PROGRAM P_Demo_FB_HVACHeatingCurve
VAR
    fb : FB_HVACHeatingCurve;                            // 被演示 FB 实例
    eDataSecurityType_in : E_HVACDataSecurityType ;
    bSetDefault_in : BOOL := FALSE;
    rOutsideTempDamped_in : REAL := 0.0;
    bDayOperation_in : BOOL := FALSE;
    bReset_in : BOOL := FALSE;
    rMinTemp_io : REAL := 0.0;
    rMaxTemp_io : REAL := 0.0;
    rNightSetback_io : REAL := 0.0;
    rTempSetpoint_Y1_io : REAL := 0.0;
    rTempSetpoint_Y2_io : REAL := 0.0;
    rTempSetpoint_Y3_io : REAL := 0.0;
    rTempSetpoint_Y4_io : REAL := 0.0;
    rOutsideTemp_X1_io : REAL := 0.0;
    rOutsideTemp_X2_io : REAL := 0.0;
    rOutsideTemp_X3_io : REAL := 0.0;
    rOutsideTemp_X4_io : REAL := 0.0;
    rTempSetpoint_out : REAL;
    bInvalidParameter_out : BOOL;
END_VAR

// ============================================================================
// Tc2_HVAC.FB_HVACHeatingCurve 演示程序
// ============================================================================
// 场景：把本 FB 实例化到一个 PLC 程序里，每周期单次调用；按需要把 VAR_INPUT 与
//       VAR_IN_OUT 接到工程信号；VAR_OUTPUT 写入对应监视变量。
// 价值：使用本 FB 比手写状态机 / 控制算法节省大量代码；与 Tc2_HVAC 体系内其它 FB
//       直接对接，命名 / 持久化 / 模式仲裁等约定一致。具体语义见 FB_HVACHeatingCurve.md 主文档。
// 验证步骤：
//   1. 右键 PLC 项目下 POUs 文件夹 → Add → Existing Item → 选本 .TcPOU 文件
//   2. 引用 Tc2_HVAC（References → Add library）
//   3. 编译 → 登录 → 运行
//   4. 在线写各 *_in 输入信号触发 FB；在线 monitor *_out 引脚观察状态
// ============================================================================

fb(
    eDataSecurityType := eDataSecurityType_in,
    bSetDefault := bSetDefault_in,
    rOutsideTempDamped := rOutsideTempDamped_in,
    bDayOperation := bDayOperation_in,
    bReset := bReset_in,
    rMinTemp := rMinTemp_io,
    rMaxTemp := rMaxTemp_io,
    rNightSetback := rNightSetback_io,
    rTempSetpoint_Y1 := rTempSetpoint_Y1_io,
    rTempSetpoint_Y2 := rTempSetpoint_Y2_io,
    rTempSetpoint_Y3 := rTempSetpoint_Y3_io,
    rTempSetpoint_Y4 := rTempSetpoint_Y4_io,
    rOutsideTemp_X1 := rOutsideTemp_X1_io,
    rOutsideTemp_X2 := rOutsideTemp_X2_io,
    rOutsideTemp_X3 := rOutsideTemp_X3_io,
    rOutsideTemp_X4 := rOutsideTemp_X4_io,
    rTempSetpoint => rTempSetpoint_out,
    bInvalidParameter => bInvalidParameter_out
);

END_PROGRAM

(* stored: Version 1.1.0.1, ProductVersion 3.1.4024.5
   POU P_Demo_FB_HVACHeatingCurve: Id {663ddc3e-7405-5011-9613-7ce8c8fa7064}, SpecialFunc None *)
